FUNCTION DEGREE_TO_RADIAN : LREAL
VAR_INPUT
	Degree : LREAL;
END_VAR

DEGREE_TO_RADIAN := Degree * (PI / 180.0);

END_FUNCTION

(* stored: Version 1.1.0.1
   POU DEGREE_TO_RADIAN: Id {1ebde5b6-531c-4aef-a1be-0aadab2b0f18}, SpecialFunc None *)
